(*
SPDX-FileCopyrightText: © 2026 Oleksandr Tiutyk <trofimich@gmail.com>
SPDX-License-Identifier: MIT
License: https://opensource.org/license/mit
*)

INTERFACE IExceptionHandler EXTENDS IObject

METHOD HandleException : BOOL
VAR_INPUT
	exception : IException;
END_VAR
END_METHOD

END_INTERFACE

(* stored: Version 1.1.0.1
   Itf IExceptionHandler: Id {b364e431-1d22-40a8-85a1-4474da6649a7}
   Method HandleException: Id {026a527f-9429-41d7-bbd6-cc7902a72610} *)
